(* PLC project Example1, KAIST_SELAB noNameNow 1.0 *)
(* stored: creationDateTime 2019-01-14T15:39:07, modificationDateTime 2019-02-19T14:21:12 *)

PROGRAM program0
  VAR
    ton1 : TON;
  END_VAR
  VAR_INPUT
    PV_OUT : INT;
    TSP : INT;
  END_VAR
  VAR_IN_OUT
    TRIP_LOGIC : BOOL;
  END_VAR
  VAR_INPUT
    K_DELAY : INT;
  END_VAR
  VAR_OUTPUT
    TON_et : INT;
  END_VAR

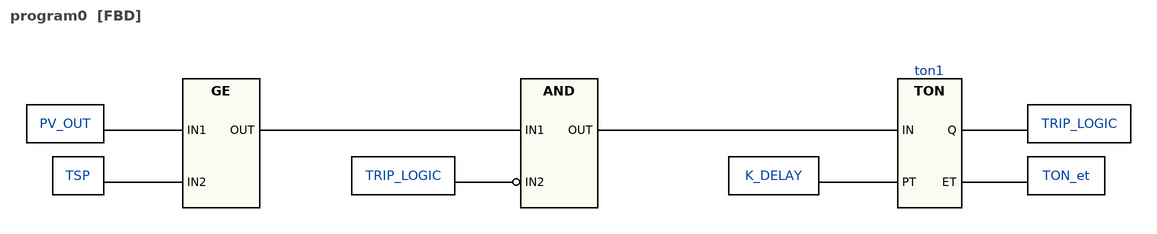
(* FBD diagram, written out as Structured Text *)
ton1(IN := PV_OUT >= TSP AND NOT TRIP_LOGIC, PT := K_DELAY);
TRIP_LOGIC := ton1.Q;
TON_et := ton1.ET;
END_PROGRAM
